// LS Electric XG5000 project: 485modbusRTU통신제어_hmi
// PLC LSPLC

PROGRAM NewProgram (task: 스캔 프로그램)

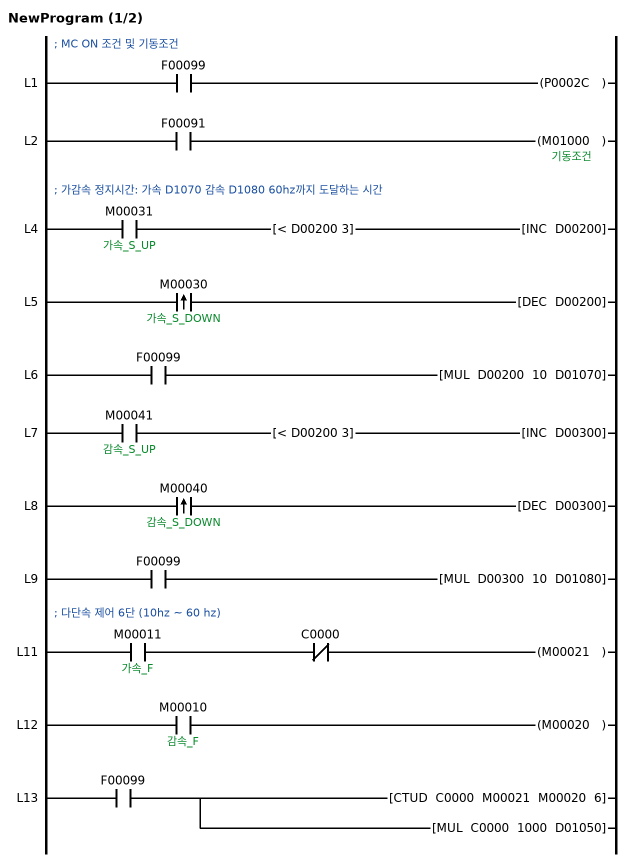
// MC ON 조건 및 기동조건
; L1
LOAD      F00099
OUT       P0002C
; L2
LOAD      F00091
OUT       M01000	// 기동조건
// 가감속 정지시간: 가속 D1070 감속 D1080 60hz까지 도달하는 시간
; L4
LOAD      M00031	// 가속_S_UP
AND<      D00200 3
INC       D00200
; L5
LOADP     M00030	// 가속_S_DOWN
DEC       D00200
; L6
LOAD      F00099
MUL       D00200 10 D01070
; L7
LOAD      M00041	// 감속_S_UP
AND<      D00200 3
INC       D00300
; L8
LOADP     M00040	// 감속_S_DOWN
DEC       D00300
; L9
LOAD      F00099
MUL       D00300 10 D01080
// 다단속 제어 6단 (10hz ~ 60 hz) 
; L11
LOAD      M00011	// 가속_F
AND NOT   C0000
OUT       M00021
; L12
LOAD      M00010	// 감속_F
OUT       M00020
; L13
LOAD      F00099
CTUD      C0000 M00021 M00020 6
MUL       C0000 1000 D01050

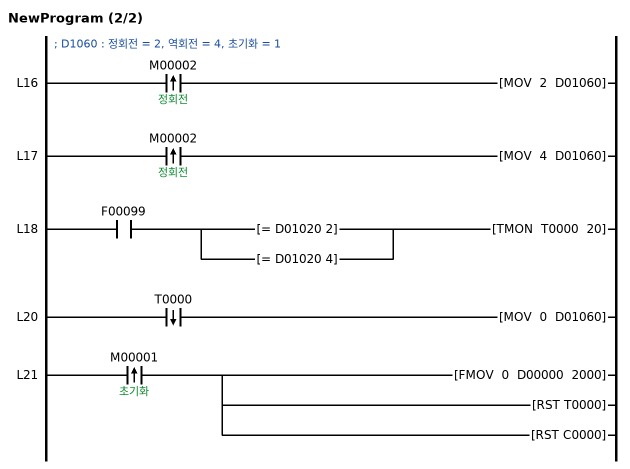
// D1060 : 정회전 = 2, 역회전 = 4, 초기화 = 1
; L16
LOADP     M00002	// 정회전
MOV       2 D01060
; L17
LOADP     M00002	// 정회전
MOV       4 D01060
; L18
LOAD      F00099
LOAD=     D01020 2
OR=       D01020 4
AND LOAD
TMON      T0000 20
; L20
LOADN     T0000
MOV       0 D01060
; L21
LOADP     M00001	// 초기화
FMOV      0 D00000 2000
RST       T0000
RST       C0000

VARIABLES AND COMMENTS (devices not used above)
M00004	BIT	역회전